TYPE ST_CalibrationInfo :
STRUCT
	iCalibrationNumber 	: UDINT;
	iUserID				: STRING(128);
	rSolventDensity 	: LREAL;
	iSolventID			: STRING(64);
	iSysMasterListRev 	: UDINT;
	iSysSettingsRev		: UDINT;
	iSolventRevision 	: UINT;
	iReplicates			: UINT;
	iAllowableFailures	: UINT;
	iCalIntervalDays	: UINT;
END_STRUCT
END_TYPE

(* stored: Version 1.1.0.1, ProductVersion 3.1.4024.15
   DUT ST_CalibrationInfo: Id {1d284007-6929-4953-badc-ac18c9b81f89} *)
